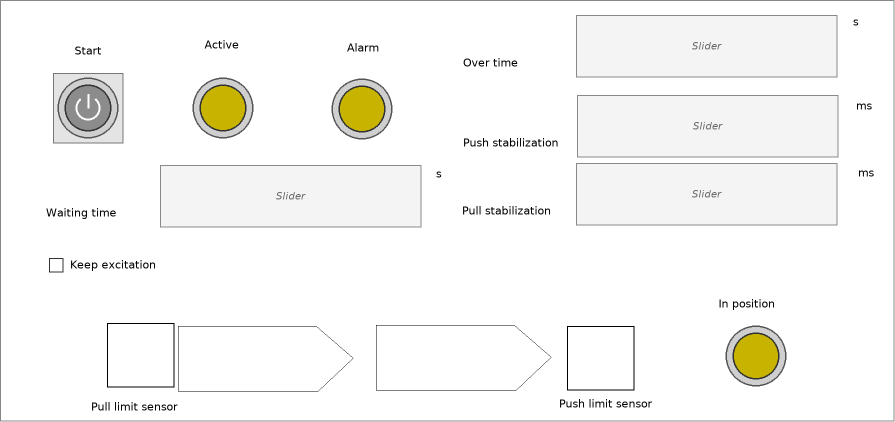
VISUALIZATION Visualization  // 895x422
    Lamp1 (188,73 70x70), variable: TargetMAIN.cylinder_1.bExecute, style: Lamp-Lamp1-Yellow
    PowerSwitch (53,73 70x70), variable: TargetMAIN.cylinder_1.bExecute, behaviour: TOGGLE, style: Switch-PowerSwitch-Gray
    Lamp1 (327,74 70x70), variable: TargetMAIN.cylinder_1.bError, style: Lamp-Lamp1-Yellow
    Slider (576,15 261x62), variable: TargetMAIN.moving_overtime, scale 0..10
    Label (460,48 150x30), "Over time"
    Slider (577,95 261x62), variable: TargetMAIN.push_stabilization, scale 0..1000
    Label (460,128 150x30), "Push stabilization"
    Label (459,196 150x30), "Pull stabilization"
    Slider (576,163 261x62), variable: TargetMAIN.pull_stabilization, scale 0..1000
    Label (43,198 150x30), "Waiting time"
    Slider (160,165 261x62), variable: TargetMAIN.stroke_interval_time, scale 0..10
    Label (288,33 150x30), "Alarm"
    Label (147,30 150x30), "Active"
    Label (13,36 150x30), "Start"
    Rectangle (107,323 67x64), colour toggle: TargetMAIN.cylinder_1_io.pull_sensor
    Rectangle (567,326 67x64), colour toggle: TargetMAIN.cylinder_1_io.push_sensor
    Label (853,91 40x30), "ms"
    Label (855,158 40x30), "ms"
    Label (850,7 40x30), "s"
    Label (433,159 40x30), "s"
    Checkbox (47,250 150x30), "Keep excitation", variable: TargetMAIN.cylinder_1.keep_actuator
    Polygon (376,325) (514,325) (551,357) (516,390) (376,390), colour toggle: TargetMAIN.cylinder_1.io.push_output
    Polygon (178,326) (316,326) (353,358) (318,391) (178,391), colour toggle: TargetMAIN.cylinder_1.io.pull_output
    Lamp1 (721,321 70x70), variable: TargetMAIN.inposition, style: Lamp-Lamp1-Yellow
    Label (672,289 150x30), "In position"
    Label (88,392 99x30), "Pull limit sensor"
    Label (556,389 99x30), "Push limit sensor"
END_VISUALIZATION

(* stored: Version 1.1.0.1, ProductVersion 3.1.4024.12
   Visu Visualization: Id {2f3bc6dd-9479-4095-b609-eb1679db70ba} *)
